TYPE E_Type_motion :
(
	eCoordonne, eMarcheArriereCoordonne, eDistance, eAngle, eCourbe 
);
END_TYPE

(* stored: Version 1.1.0.1, ProductVersion 3.1.4024.11
   DUT E_Type_motion: Id {2ae8d345-f9b0-49b5-9d8f-dd053471f6b7} *)
